TYPE TcoInterpolatorStatus :
STRUCT
	ActionDescription : STRING(100);
	AlarmMessage : STRING(254);	
	Progress:int;
	Data: TcoGenericInterpolatorData;
END_STRUCT
END_TYPE

(* stored: Version 1.1.0.1, ProductVersion 3.1.4024.12
   DUT TcoInterpolatorStatus: Id {81c7f655-c138-020f-36f0-7ec088e0d95d} *)
